{attribute 'GeneratedUsingTerminal: KL6831'}
{attribute addProperty BoxType "KL6831"}
{attribute addProperty Description ""}
{attribute addProperty Physics ""}
{attribute addProperty Id "Channel_1AT %Q*Channel_A1C14FB40"}
{attribute addProperty CRC "3193527458"}
{attribute addProperty Size "0"}
TYPE KL6831_BE595CA2 :
STRUCT
	{attribute addProperty Name "Channel_1"}
	Channel_1 : Channel_A1C14FB4;
END_STRUCT
END_TYPE

(* stored: Version 1.2.0.0, ProductVersion 3.1.4024.9
   DUT KL6831_BE595CA2: Id {2110050d-f12f-4e15-8aa0-d969bb421930} *)
